{attribute 'no_explicit_call' := 'do not call this POU directly'} 
FUNCTION_BLOCK CRC IMPLEMENTS Tc3_AlgoInterfaces.IDigest
VAR
	// values are precalulated in FB_Init 
	CRCTableInitialized				: BOOL;
	// Precalcated lookup table
	CRC_Table 						: ARRAY[0..TABLESIZE-1] OF XWORD;
	// Current crc
	currentCrc						: XWORD;					
	// CRC parameters
	_crcType						: E_CRC_TYPE;
	_polynomial						: XWORD;		// polynomial 
	_polynomial_					: XWORD;		// reflected polynomial 
	_bitWidth						: BYTE;
	_initCrc						: XWORD;
	_reflectInitial					: BOOL;
	_reflected						: BOOL;
	_xorOut							: XWORD;
	_check							: XWORD;
	_residue						: XWORD;
	// internal 
	isInitialReflected				: BOOL;
END_VAR
VAR CONSTANT
	// Maximum size of the lookup table (no of byte values)
	TABLESIZE						: UINT := 256;
END_VAR

// use compute method

PROPERTY algorithm : STRING
GET
algorithm := TO_STRING(_crcType);
END_GET
END_PROPERTY

// Computes CRC using a standard (non-reflected) lookup table
METHOD PRIVATE computeNormal : XWORD
VAR_INPUT
    pData 						: POINTER TO BYTE;
	dataSize					: DWORD;
END_VAR
VAR
	pByte 						: POINTER TO BYTE;
	bByte						: BYTE;
	mode 						: BYTE;
	i 							: DWORD;
	lookupIndex					: BYTE;
END_VAR
mode					:= TO_BYTE(_bitWidth / 8) - 1;
computeNormal 			:= currentCrc;

pByte					:= pData;
FOR i := 0 TO dataSize - 1 DO
	bByte				:= pByte^;
	pByte				:= pByte + 1;
	lookupIndex			:= TO_BYTE(SHR(computeNormal, GVC_CRC.crcShift[mode]) XOR bByte);	
	IF (mode = E_CRC_Mode.CRC8)	THEN
		computeNormal	:= CRC_Table[lookupIndex];
	ELSE
		computeNormal	:= SHL(computeNormal, 8) XOR CRC_Table[lookupIndex];
	END_IF
	computeNormal		:= computeNormal AND GVC_CRC.crcMasks[mode]; 
END_FOR
END_METHOD

// Computes CRC using a reflected lookup table
METHOD PRIVATE computeReflected : XWORD
VAR_INPUT
    pData 						: POINTER TO BYTE;
	dataSize					: DWORD;
END_VAR
VAR
	pByte 						: POINTER TO BYTE;
	bByte						: BYTE;
	i 							: DWORD;
	lookupIndex					: BYTE;
END_VAR
computeReflected 		:= currentCrc;

pByte					:= pData;
FOR i := 0 TO dataSize - 1 DO
	bByte				:= pByte^;
	pByte				:= pByte + 1;
	lookupIndex			:= TO_BYTE((computeReflected XOR bByte) AND GVC_CRC.crcMasks[0]);
	computeReflected	:= SHR(computeReflected, 8) XOR CRC_Table[lookupIndex];
END_FOR
END_METHOD

METHOD FB_Init: BOOL
VAR_INPUT
    bInitRetains				: BOOL; // TRUE: the retain variables are initialized (reset warm / reset cold)
    bInCopyCode					: BOOL; // TRUE: the instance will be copied to the copy code afterward (online change)   
	crcType						: E_CRC_TYPE;
END_VAR
// Pass to the local init
reconfigure(crcType);
END_METHOD

(* Finalize the input and return any number of output bytes.*)
METHOD finalize
VAR_IN_OUT
	out					: ARRAY [*] OF BYTE;
END_VAR
VAR
	byteVal, mode		: BYTE;
	i, j, ub			: DINT;
END_VAR
// Final xor and mask
mode					:= TO_BYTE(_bitWidth / 8) - 1;
currentCrc				:= (currentCrc XOR _xorOut) AND GVC_CRC.crcMasks[mode];

j 	:= LOWER_BOUND(out, 1);
ub 	:= UPPER_BOUND(out, 1);
FOR i := 0 TO GVC_CRC.CRC_Parameters[_crcType].bitWidth / 8 - 1 DO
	IF i > ub THEN // in case the wrong crc result container was passed
		EXIT;
	ELSE
		byteVal	:= TO_BYTE(SHR(currentCrc, i * 8));
		//byteVal := TO_BYTE(SHR(byteVal, 56)
		out[i]  := byteVal; // TO_BYTE(SHR(SHL(currentCrc, i * 8), 56));
	END_IF
END_FOR
END_METHOD

// Generates a standard CRC lookup table
METHOD PRIVATE generateNormalCRCTable : BOOL
VAR
	mode					: BYTE;
	crc						: XWORD;
	i, j					: UINT; 
END_VAR
generateNormalCRCTable := FALSE;
mode := (_bitWidth / 8) - 1;

FOR i := 0 TO TABLESIZE - 1 DO
	crc			:= (SHL(TO___XWORD(i), GVC_CRC.CRCShift[mode])) AND GVC_CRC.CRCMasks[mode];
	FOR j := 0 TO 7 DO
		IF (crc AND GVC_CRC.CRCMsb[Mode]) = 0 THEN
			crc :=  SHL(crc, 1); 
		ELSE
			crc := SHL(crc, 1) XOR _polynomial;
		END_IF
		crc		:= crc AND GVC_CRC.CRCMasks[mode];
  	END_FOR
	CRC_Table[i]:= crc;
END_FOR
generateNormalCRCTable := TRUE;
END_METHOD

// Generates a reflected CRC lookup table
METHOD PRIVATE generateReflectedCRCTable : BOOL
VAR
	mode					: BYTE;
	crc						: XWORD;
	i, j					: UINT; 
END_VAR
generateReflectedCRCTable := FALSE;	 
mode := (_bitWidth / 8) - 1;

FOR i := 0 TO TABLESIZE - 1 DO
	crc			:= i;
	FOR j := 0 TO 7 DO
		IF (crc AND 16#1) = 0 THEN
			crc :=  SHR(crc, 1); 
		ELSE
			crc := SHR(crc, 1) XOR _polynomial_;
		END_IF
		crc		:= crc AND GVC_CRC.CRCMasks[mode];
  	END_FOR
	CRC_Table[i]:= crc;
END_FOR
generateReflectedCRCTable := TRUE;
END_METHOD

METHOD init
// Reset the crc to the configured initial value 
currentCrc 			:= _initCrc;
isInitialReflected		:= FALSE;
END_METHOD

// Reconfigures and initializes the CRC table in function of chosen CRC Type
METHOD reconfigure : bool
VAR_INPUT
	crcType						: E_CRC_TYPE;
END_VAR
// CRC parameters
_crcType				:= crcType;
_bitWidth				:= GVC_CRC.CRC_Parameters[_crcType].bitWidth;
_polynomial				:= GVC_CRC.CRC_Parameters[_crcType].polynomial; 
_polynomial_			:= reflectBits(_polynomial, _bitWidth);
_initCrc				:= GVC_CRC.CRC_Parameters[_crcType].initCRC;
_reflectInitial			:= GVC_CRC.CRC_Parameters[_crcType].reflectInitial;
_reflected				:= GVC_CRC.CRC_Parameters[_crcType].reflected;
_xorOut					:= GVC_CRC.CRC_Parameters[_crcType].xorOut;
_check					:= GVC_CRC.CRC_Parameters[_crcType].check;
_residue				:= GVC_CRC.CRC_Parameters[_crcType].residue;

// Build CRC table
CRCTableInitialized := FALSE;
IF GVC_CRC.CRC_Parameters[_crcType].polynomial > 0 THEN		// Valid polynomial
	IF _reflected			THEN
		CRCTableInitialized	:= generateReflectedCRCTable();
	ELSE
		CRCTableInitialized	:= generateNormalCRCTable();
	END_IF
END_IF

// initialize 
init();
END_METHOD

// Reflects the bit order of a value
METHOD PRIVATE reflectBits		: XWORD
VAR_INPUT
	value 						: XWORD;
	bitWidth					: BYTE;
END_VAR
VAR
	i							: BYTE;
	shrValue					: XWORD;
	andBit						: XWORD;
END_VAR
reflectBits 		:= 16#0;
shrValue 		:= value;
andBit 			:= shrValue AND 16#1;
reflectBits 		:= reflectBits + andBit;
FOR i := 1 TO bitWidth - 1 DO
	reflectBits 	:= SHL(reflectBits,1);
	shrValue 	:= SHR(shrValue,1);
	andBit 		:= shrValue AND 16#1;
	reflectBits 	:= reflectBits + andBit;
END_FOR
END_METHOD

(* Add input, depending on the algorithm this could be called any number of times.*)
METHOD update
VAR_INPUT
	input						: POINTER TO BYTE;
	input_len					: DWORD;
END_VAR
IF _reflectInitial		AND NOT 
	isInitialReflected		THEN
	currentCrc			:= reflectBits(currentCrc, _bitWidth);
	isInitialReflected		:= TRUE;
END_IF

IF _reflected			THEN
	currentCrc := computeReflected(input, input_len);
ELSE
	currentCrc := computeNormal(input, input_len);
END_IF
END_METHOD

END_FUNCTION_BLOCK

(* stored: Version 1.1.0.1
   POU CRC: Id {ae31b935-10b3-41d4-a99d-e381a90ecc2f}, SpecialFunc None
   Property algorithm: Id {1162413a-937e-404d-a892-a75645792905}
   Get Get: Id {87cf8149-c304-4d20-8aa3-ef9ac26e26d2}
   Method computeNormal: Id {ef873984-0c49-471a-bff4-77b5bfcd3425}
   Method computeReflected: Id {734aecd5-6748-4cb2-8d3a-5f148b24b568}
   Method FB_Init: Id {c3277821-a481-40ce-beed-521fc383580f}
   Method finalize: Id {bd24b3a6-ebfe-4f8f-ade8-44898b1b0c91}
   Method generateNormalCRCTable: Id {6c6ace14-5f31-4b1d-8edd-32bfdb419666}
   Method generateReflectedCRCTable: Id {6fd1f359-95af-457f-859f-8cc00ef7118c}
   Method init: Id {a8faa941-fa55-4d21-b331-67b8d2c894c6}
   Method reconfigure: Id {6eeda4d7-cd42-4d47-baf7-fda5eed4329f}
   Method reflectBits: Id {2aab224d-daf4-4902-adf3-77404855cc06}
   Method update: Id {8a3da472-876d-4a34-988a-304389337cb5} *)
